FUNCTION_BLOCK FB_FuseAdvanced 
VAR_INPUT
END_VAR
VAR_OUTPUT
END_VAR
VAR
	Chn1 : EL922x_ChannelExtended;
	Chn2 : EL922x_ChannelExtended;
END_VAR

END_FUNCTION_BLOCK

(* stored: Version 1.1.0.1, ProductVersion 3.1.4024.5
   POU FB_FuseAdvanced: Id {e62c69d5-30eb-4744-8257-2617f7fd3e98}, SpecialFunc None *)
